// TIA Portal V20 export
// export: Created 2026-07-12T13:33:04.7141366Z, ExportSetting WithDefaults, DisplayName Totally Integrated Automation Portal, DisplayVersion V20 Update 4, DisplayName TIA Portal Openness, DisplayVersion V20 Update 4, DisplayName TIA Portal Version Control Interface, DisplayVersion V20 Update 4, DisplayName STEP 7 Professional, DisplayVersion V20 Update 4, DisplayName STEP 7 Safety, DisplayVersion V20 Update 2, DisplayName WinCC Basic/Comfort/Advanced, DisplayVersion V20 Update 4, DisplayName WinCC Unified, DisplayVersion V20 Update 4
DATA_BLOCK "DB_fieldDevices"   // DB3
{ S7_Optimized_Access := 'FALSE' }
VERSION : 0.1
// stored: AutoNumber true, IsOnlyStoredInLoadMemory false, IsWriteProtectedInAS false
   VAR RETAIN
      StartStop_Cmd : Bool;
      Reset : Bool;
      L_CutlineSensor : Array[1..15] of Bool;
      B_CutlineButtons : Array[1..15] of Bool;
      B_Controls : Array[1..15] of Bool;
   END_VAR
BEGIN
   // L_CutlineSensor[1] : 00
   // L_CutlineSensor[2] : 30
   // L_CutlineSensor[3] : 36
   // L_CutlineSensor[4] : 42
   // L_CutlineSensor[5] : 48
   // L_CutlineSensor[6] : 54
   // L_CutlineSensor[7] : 60
   // L_CutlineSensor[8] : 66
   // B_Controls[1] : Start/Stop
   // B_Controls[2] : Reset
END_DATA_BLOCK
